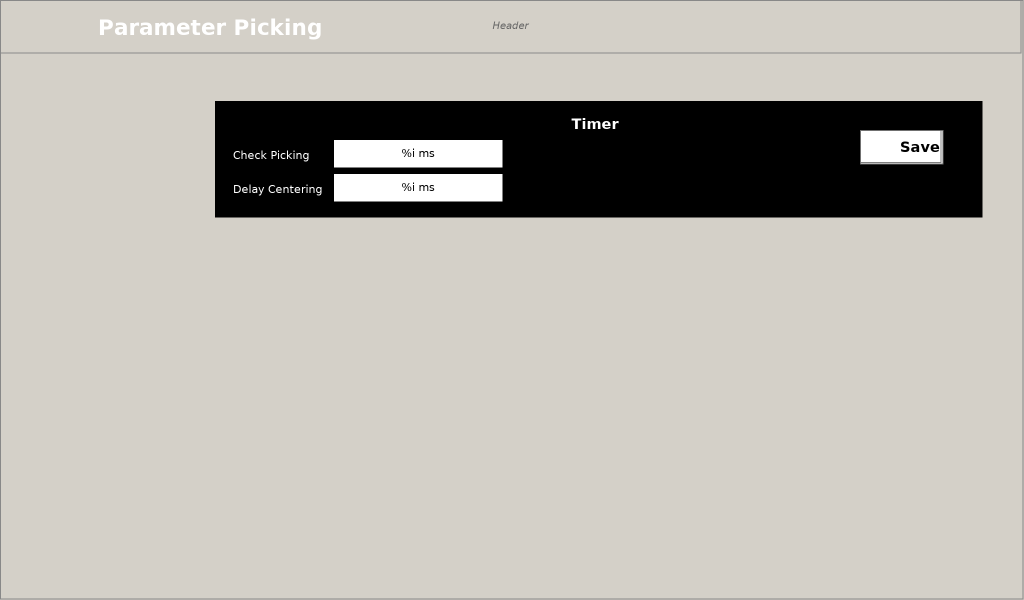
VISUALIZATION MPicking  // 1024x600
    Frame (0,-2 1021x55)
        shows Header()
    Label (95,15 250x25), "Parameter Picking"
    RoundedRectangle (215,101 767x116)
    Label (243,104 704x40), "Timer"
    Label (230,138 103x35), "Check Picking"
    RoundedRectangle (333,139 170x29), "%i ms", text variable: HMI_GVL.Tmr_Picking
        OnMouseClick: write the text variable via Default
    Button (860,130 83x34), "Save", image: VisuSymbols.Symbols.Save
        tap InputOutput_GVL.TestMode[100]
    Label (230,172 104x35), "Delay Centering"
    RoundedRectangle (333,173 170x29), "%i ms", text variable: HMI_GVL.Tmr_Centering
        OnMouseClick: write the text variable via Default
END_VISUALIZATION

(* stored: Version 1.1.0.1, ProductVersion 3.1.4024.12
   Visu MPicking: Id {4b8336de-f889-44d7-ac43-c8a1b12da873} *)
